REGION Network 26: Signal conditioning — Consolidate the auto or manual state request
   // ▀▀▀▀▀▀▀▀▀▀▀▀▀▀▀▀▀▀▀▀▀▀▀▀▀▀▀▀▀▀▀▀▀▀▀▀▀▀▀▀▀▀▀▀
   // Determine the valve state required by the automatic/manual mode selection:
   // 
   //    1.  If manual mode is active set wrkCtrlAutManOpCl to match the current manual 
   //      mode requested state (ctrl_Man_OpenClose)
   // 
   //    2.  If automatic mode is active set wrkCtrlAutManOpCl to match the current automatic 
   //      mode requested state (ctrl_Aut_OpenClose)
   // ▄▄▄▄▄▄▄▄▄▄▄▄▄▄▄▄▄▄▄▄▄▄▄▄▄▄▄▄▄▄▄▄▄▄▄▄▄▄▄▄▄▄▄▄
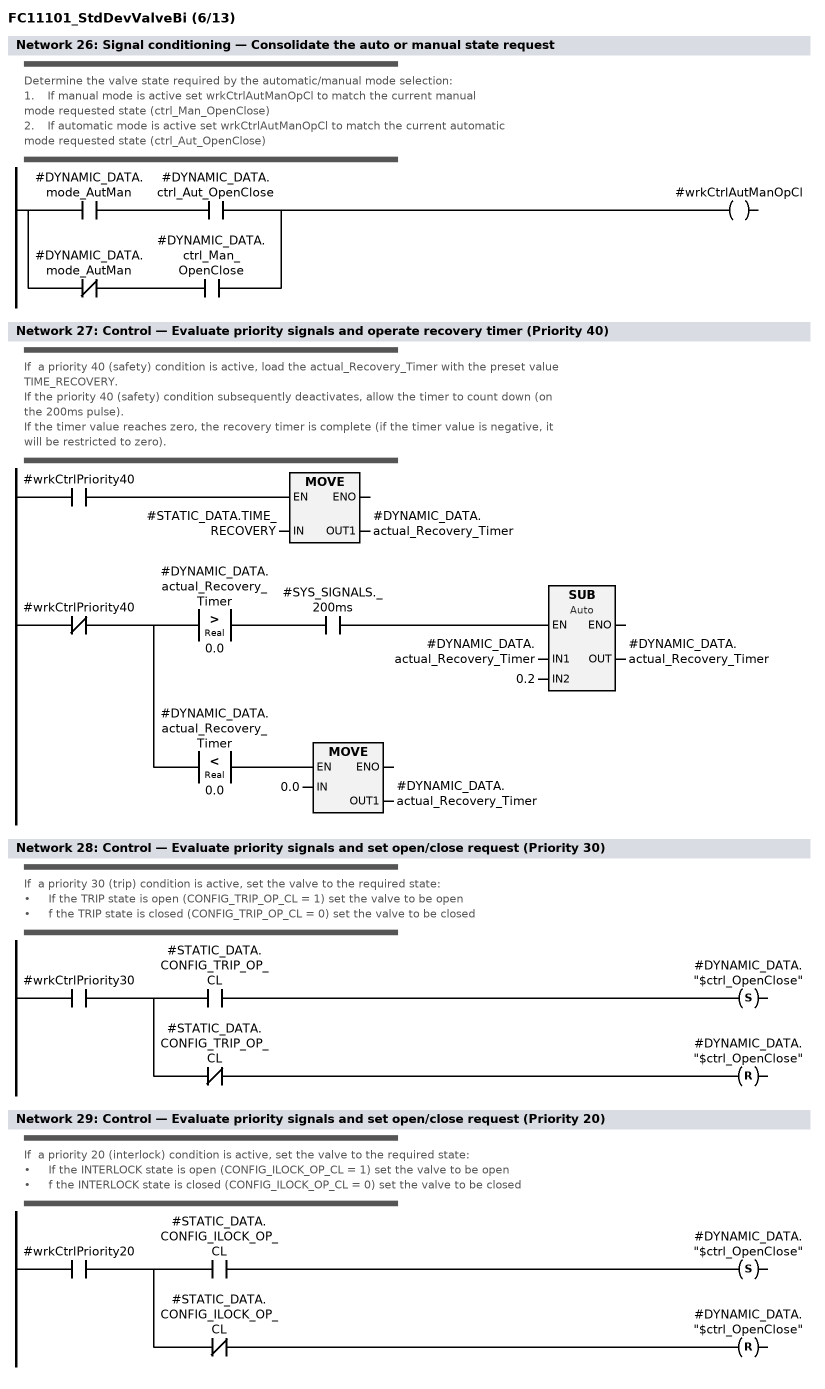
   RUNG wire#powerrail
      Contact( #DYNAMIC_DATA.mode_AutMan )
      Contact( #DYNAMIC_DATA.ctrl_Aut_OpenClose )
      wire#w1
      Coil( #wrkCtrlAutManOpCl )
   END_RUNG
   RUNG wire#powerrail
      I_Contact( #DYNAMIC_DATA.mode_AutMan )
      Contact( #DYNAMIC_DATA.ctrl_Man_OpenClose )
   END_RUNG wire#w1
   // the same network as SCL:
   #wrkCtrlAutManOpCl := (#DYNAMIC_DATA.mode_AutMan AND #DYNAMIC_DATA.ctrl_Aut_OpenClose) OR (NOT #DYNAMIC_DATA.mode_AutMan AND #DYNAMIC_DATA.ctrl_Man_OpenClose);
END_REGION

REGION Network 27: Control — Evaluate priority signals and operate recovery timer (Priority 40)
   // ▀▀▀▀▀▀▀▀▀▀▀▀▀▀▀▀▀▀▀▀▀▀▀▀▀▀▀▀▀▀▀▀▀▀▀▀▀▀▀▀▀▀▀▀
   // If  a priority 40 (safety) condition is active, load the actual_Recovery_Timer with the preset value 
   // TIME_RECOVERY.
   // 
   // If the priority 40 (safety) condition subsequently deactivates, allow the timer to count down (on 
   // the 200ms pulse).
   // 
   // If the timer value reaches zero, the recovery timer is complete (if the timer value is negative, it
   // will be restricted to zero).
   // ▄▄▄▄▄▄▄▄▄▄▄▄▄▄▄▄▄▄▄▄▄▄▄▄▄▄▄▄▄▄▄▄▄▄▄▄▄▄▄▄▄▄▄▄
   RUNG wire#powerrail
      Contact( #wrkCtrlPriority40 )
      Move(in := #STATIC_DATA.TIME_RECOVERY, out1 => #DYNAMIC_DATA.actual_Recovery_Timer)
   END_RUNG
   RUNG wire#powerrail
      I_Contact( #wrkCtrlPriority40 )
      wire#w1
      { S7_Templates := "SrcType := Real" } GT_Contact(in1 := #DYNAMIC_DATA.actual_Recovery_Timer, in2 := 0.0)
      Contact( #SYS_SIGNALS._200ms )
      Sub(in1 := #DYNAMIC_DATA.actual_Recovery_Timer, in2 := 0.2, out => #DYNAMIC_DATA.actual_Recovery_Timer)
   END_RUNG
   RUNG wire#w1
      { S7_Templates := "SrcType := Real" } LT_Contact(in1 := #DYNAMIC_DATA.actual_Recovery_Timer, in2 := 0.0)
      Move(in := 0.0, out1 => #DYNAMIC_DATA.actual_Recovery_Timer)
   END_RUNG
   // the same network as SCL:
   IF #wrkCtrlPriority40 THEN #DYNAMIC_DATA.actual_Recovery_Timer := #STATIC_DATA.TIME_RECOVERY; END_IF;
   IF NOT #wrkCtrlPriority40 AND (#DYNAMIC_DATA.actual_Recovery_Timer > 0.0) AND #SYS_SIGNALS._200ms THEN
       #DYNAMIC_DATA.actual_Recovery_Timer := #DYNAMIC_DATA.actual_Recovery_Timer - 0.2;
   END_IF;
   IF NOT #wrkCtrlPriority40 AND (#DYNAMIC_DATA.actual_Recovery_Timer < 0.0) THEN
       #DYNAMIC_DATA.actual_Recovery_Timer := 0.0;
   END_IF;
END_REGION

REGION Network 28: Control — Evaluate priority signals and set open/close request (Priority 30)
   // ▀▀▀▀▀▀▀▀▀▀▀▀▀▀▀▀▀▀▀▀▀▀▀▀▀▀▀▀▀▀▀▀▀▀▀▀▀▀▀▀▀▀▀▀
   // If  a priority 30 (trip) condition is active, set the valve to the required state:
   // 
   //    •   If the TRIP state is open (CONFIG_TRIP_OP_CL = 1) set the valve to be open
   // 
   //    •   f the TRIP state is closed (CONFIG_TRIP_OP_CL = 0) set the valve to be closed
   // ▄▄▄▄▄▄▄▄▄▄▄▄▄▄▄▄▄▄▄▄▄▄▄▄▄▄▄▄▄▄▄▄▄▄▄▄▄▄▄▄▄▄▄▄
   RUNG wire#powerrail
      Contact( #wrkCtrlPriority30 )
      wire#w1
      Contact( #STATIC_DATA.CONFIG_TRIP_OP_CL )
      S_Coil( #DYNAMIC_DATA."$ctrl_OpenClose" )
   END_RUNG
   RUNG wire#w1
      I_Contact( #STATIC_DATA.CONFIG_TRIP_OP_CL )
      R_Coil( #DYNAMIC_DATA."$ctrl_OpenClose" )
   END_RUNG
   // the same network as SCL:
   IF #wrkCtrlPriority30 AND #STATIC_DATA.CONFIG_TRIP_OP_CL THEN
       #DYNAMIC_DATA."$ctrl_OpenClose" := TRUE;
   END_IF;
   IF #wrkCtrlPriority30 AND NOT #STATIC_DATA.CONFIG_TRIP_OP_CL THEN
       #DYNAMIC_DATA."$ctrl_OpenClose" := FALSE;
   END_IF;
END_REGION

REGION Network 29: Control — Evaluate priority signals and set open/close request (Priority 20)
   // ▀▀▀▀▀▀▀▀▀▀▀▀▀▀▀▀▀▀▀▀▀▀▀▀▀▀▀▀▀▀▀▀▀▀▀▀▀▀▀▀▀▀▀▀
   // If  a priority 20 (interlock) condition is active, set the valve to the required state:
   // 
   //    •   If the INTERLOCK state is open (CONFIG_ILOCK_OP_CL = 1) set the valve to be open
   // 
   //    •   f the INTERLOCK state is closed (CONFIG_ILOCK_OP_CL = 0) set the valve to be closed
   // ▄▄▄▄▄▄▄▄▄▄▄▄▄▄▄▄▄▄▄▄▄▄▄▄▄▄▄▄▄▄▄▄▄▄▄▄▄▄▄▄▄▄▄▄
   RUNG wire#powerrail
      Contact( #wrkCtrlPriority20 )
      wire#w1
      Contact( #STATIC_DATA.CONFIG_ILOCK_OP_CL )
      S_Coil( #DYNAMIC_DATA."$ctrl_OpenClose" )
   END_RUNG
   RUNG wire#w1
      I_Contact( #STATIC_DATA.CONFIG_ILOCK_OP_CL )
      R_Coil( #DYNAMIC_DATA."$ctrl_OpenClose" )
   END_RUNG
   // the same network as SCL:
   IF #wrkCtrlPriority20 AND #STATIC_DATA.CONFIG_ILOCK_OP_CL THEN
       #DYNAMIC_DATA."$ctrl_OpenClose" := TRUE;
   END_IF;
   IF #wrkCtrlPriority20 AND NOT #STATIC_DATA.CONFIG_ILOCK_OP_CL THEN
       #DYNAMIC_DATA."$ctrl_OpenClose" := FALSE;
   END_IF;
END_REGION

REGION Network 30: Control — Evaluate priority signals and set open/close request (Priority 10)
   // ▀▀▀▀▀▀▀▀▀▀▀▀▀▀▀▀▀▀▀▀▀▀▀▀▀▀▀▀▀▀▀▀▀▀▀▀▀▀▀▀▀▀▀▀
   // If  a priority 10 (permissive) condition is active, set the valve to the required state:
   // 
   // 
   // PERMITTED STATE IS OPEN — CONDITIONS:
   // 
   //    •   If the Permitted state is open and Aut/Man request is for open, 
   //      set the valve to be open [Branch 1]
   // 
   //    •   If the Permitted state is open and Aut/Man request is for closed, and the current
   //      valve output matches this state (closed), set the valve to be closed (maintain the
   //      current state) [Branch 6]
   // 
   //    •   If the Permitted state is open and Aut/Man request is for closed, and the current
   //      valve output matches the open state, set the valve to be open (override the
   //      auto/man request [Branch 2]
   // 
   // PERMITTED STATE IS CLOSED — CONDITIONS:
   // 
   //    •   If the Permitted state is closed and Aut/Man request is for closed,
   //      set the valve to be  closed [Branch 4]
   // 
   //    •   If the Permitted state is closed and Aut/Man request is for open, and the current
   //      valve output matches this state (open), set the valve to be open (maintain the
   //      current state) [Branch 3]
   // 
   //    •   If the Permitted state is closed and Aut/Man request is for open, and the current
   //      valve output matches the closed state, set the valve to be closed (override the
   //      auto/man request [Branch 5]
   // ▄▄▄▄▄▄▄▄▄▄▄▄▄▄▄▄▄▄▄▄▄▄▄▄▄▄▄▄▄▄▄▄▄▄▄▄▄▄▄▄▄▄▄▄
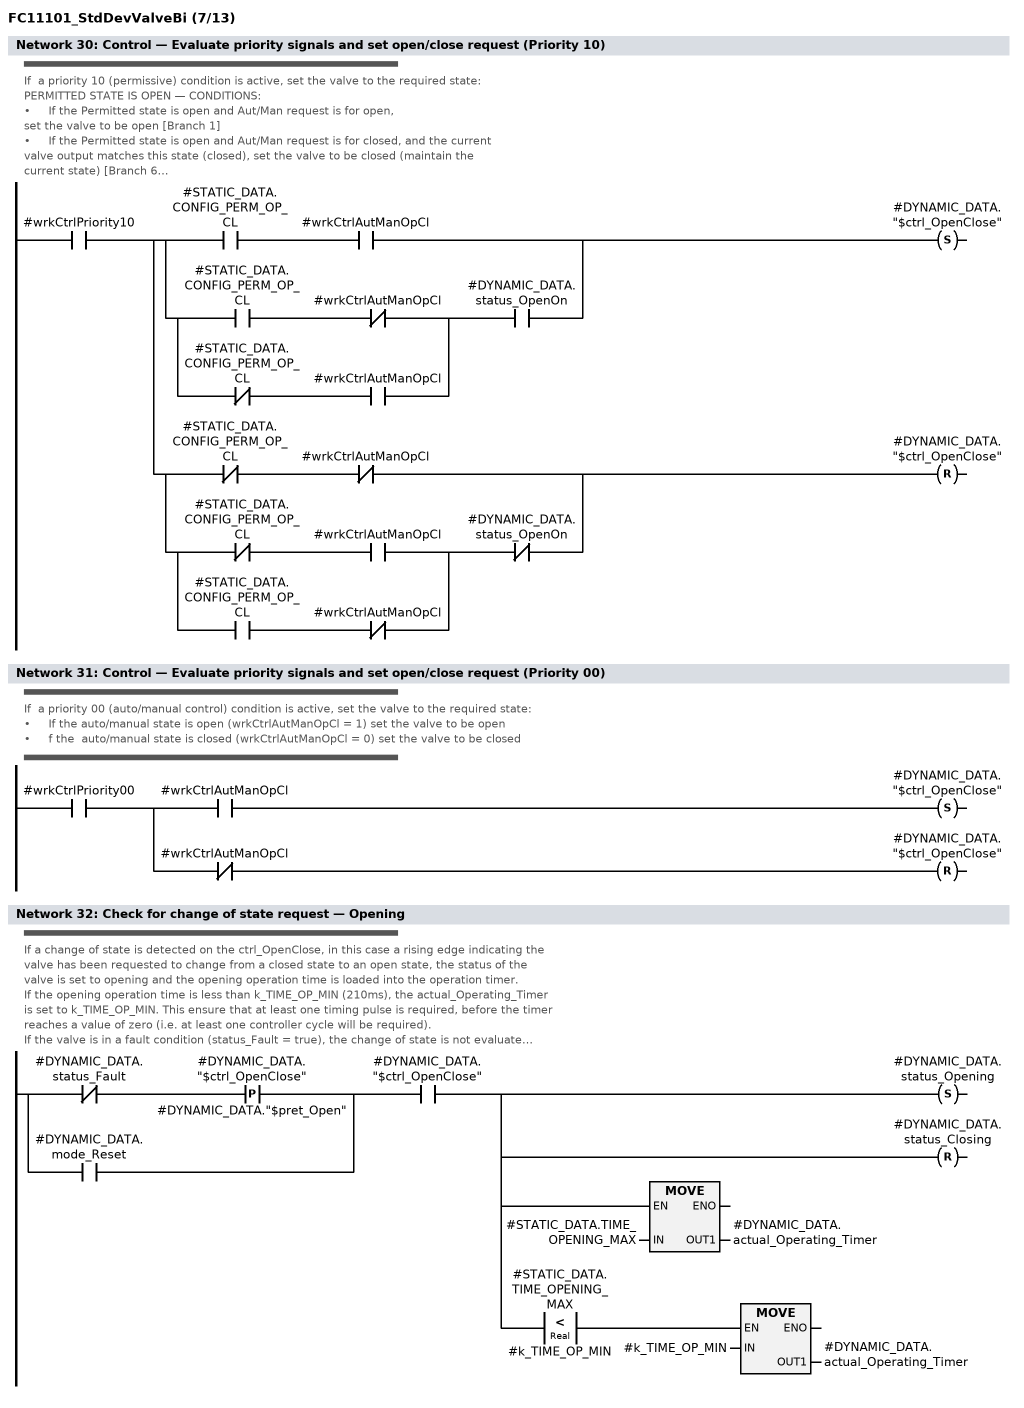
   RUNG wire#powerrail
      Contact( #wrkCtrlPriority10 )
      wire#w1
      Contact( #STATIC_DATA.CONFIG_PERM_OP_CL )
      Contact( #wrkCtrlAutManOpCl )
      wire#w2
      S_Coil( #DYNAMIC_DATA."$ctrl_OpenClose" )
   END_RUNG
   RUNG wire#w1
      Contact( #STATIC_DATA.CONFIG_PERM_OP_CL )
      I_Contact( #wrkCtrlAutManOpCl )
      wire#w3
      Contact( #DYNAMIC_DATA.status_OpenOn )
   END_RUNG wire#w2
   RUNG wire#w1
      I_Contact( #STATIC_DATA.CONFIG_PERM_OP_CL )
      Contact( #wrkCtrlAutManOpCl )
   END_RUNG wire#w3
   RUNG wire#w1
      I_Contact( #STATIC_DATA.CONFIG_PERM_OP_CL )
      I_Contact( #wrkCtrlAutManOpCl )
      wire#w4
      R_Coil( #DYNAMIC_DATA."$ctrl_OpenClose" )
   END_RUNG
   RUNG wire#w1
      I_Contact( #STATIC_DATA.CONFIG_PERM_OP_CL )
      Contact( #wrkCtrlAutManOpCl )
      wire#w5
      I_Contact( #DYNAMIC_DATA.status_OpenOn )
   END_RUNG wire#w4
   RUNG wire#w1
      Contact( #STATIC_DATA.CONFIG_PERM_OP_CL )
      I_Contact( #wrkCtrlAutManOpCl )
   END_RUNG wire#w5
   // the same network as SCL:
   IF #wrkCtrlPriority10 AND ((#STATIC_DATA.CONFIG_PERM_OP_CL AND #wrkCtrlAutManOpCl) OR (((#STATIC_DATA.CONFIG_PERM_OP_CL AND NOT #wrkCtrlAutManOpCl) OR (NOT #STATIC_DATA.CONFIG_PERM_OP_CL AND #wrkCtrlAutManOpCl)) AND #DYNAMIC_DATA.status_OpenOn)) THEN
       #DYNAMIC_DATA."$ctrl_OpenClose" := TRUE;
   END_IF;
   IF #wrkCtrlPriority10 AND ((NOT #STATIC_DATA.CONFIG_PERM_OP_CL AND NOT #wrkCtrlAutManOpCl) OR (((NOT #STATIC_DATA.CONFIG_PERM_OP_CL AND #wrkCtrlAutManOpCl) OR (#STATIC_DATA.CONFIG_PERM_OP_CL AND NOT #wrkCtrlAutManOpCl)) AND NOT #DYNAMIC_DATA.status_OpenOn)) THEN
       #DYNAMIC_DATA."$ctrl_OpenClose" := FALSE;
   END_IF;
END_REGION

REGION Network 31: Control — Evaluate priority signals and set open/close request (Priority 00)
   // ▀▀▀▀▀▀▀▀▀▀▀▀▀▀▀▀▀▀▀▀▀▀▀▀▀▀▀▀▀▀▀▀▀▀▀▀▀▀▀▀▀▀▀▀
   // If  a priority 00 (auto/manual control) condition is active, set the valve to the required state:
   // 
   //    •   If the auto/manual state is open (wrkCtrlAutManOpCl = 1) set the valve to be open
   // 
   //    •   f the  auto/manual state is closed (wrkCtrlAutManOpCl = 0) set the valve to be closed
   // ▄▄▄▄▄▄▄▄▄▄▄▄▄▄▄▄▄▄▄▄▄▄▄▄▄▄▄▄▄▄▄▄▄▄▄▄▄▄▄▄▄▄▄▄
   RUNG wire#powerrail
      Contact( #wrkCtrlPriority00 )
      wire#w1
      Contact( #wrkCtrlAutManOpCl )
      S_Coil( #DYNAMIC_DATA."$ctrl_OpenClose" )
   END_RUNG
   RUNG wire#w1
      I_Contact( #wrkCtrlAutManOpCl )
      R_Coil( #DYNAMIC_DATA."$ctrl_OpenClose" )
   END_RUNG
   // the same network as SCL:
   IF #wrkCtrlPriority00 AND #wrkCtrlAutManOpCl THEN #DYNAMIC_DATA."$ctrl_OpenClose" := TRUE; END_IF;
   IF #wrkCtrlPriority00 AND NOT #wrkCtrlAutManOpCl THEN #DYNAMIC_DATA."$ctrl_OpenClose" := FALSE; END_IF;
END_REGION

REGION Network 32: Check for change of state request — Opening
   // ▀▀▀▀▀▀▀▀▀▀▀▀▀▀▀▀▀▀▀▀▀▀▀▀▀▀▀▀▀▀▀▀▀▀▀▀▀▀▀▀▀▀▀▀
   // If a change of state is detected on the ctrl_OpenClose, in this case a rising edge indicating the
   // valve has been requested to change from a closed state to an open state, the status of the
   // valve is set to opening and the opening operation time is loaded into the operation timer.
   // 
   // If the opening operation time is less than k_TIME_OP_MIN (210ms), the actual_Operating_Timer 
   // is set to k_TIME_OP_MIN. This ensure that at least one timing pulse is required, before the timer 
   // reaches a value of zero (i.e. at least one controller cycle will be required).
   // 
   // If the valve is in a fault condition (status_Fault = true), the change of state is not evaluated
   // until the fault condition has cleared
   // 
   // Note: the timer is also triggered if the Reset signal is received and the valve is requested open.
   // ▄▄▄▄▄▄▄▄▄▄▄▄▄▄▄▄▄▄▄▄▄▄▄▄▄▄▄▄▄▄▄▄▄▄▄▄▄▄▄▄▄▄▄▄
   RUNG wire#powerrail
      I_Contact( #DYNAMIC_DATA.status_Fault )
      P_Contact(operand := #DYNAMIC_DATA."$ctrl_OpenClose", bit := #DYNAMIC_DATA."$pret_Open")
      wire#w1
      Contact( #DYNAMIC_DATA."$ctrl_OpenClose" )
      wire#w2
      S_Coil( #DYNAMIC_DATA.status_Opening )
   END_RUNG
   RUNG wire#powerrail
      Contact( #DYNAMIC_DATA.mode_Reset )
   END_RUNG wire#w1
   RUNG wire#w2
      R_Coil( #DYNAMIC_DATA.status_Closing )
   END_RUNG
   RUNG wire#w2
      Move(in := #STATIC_DATA.TIME_OPENING_MAX, out1 => #DYNAMIC_DATA.actual_Operating_Timer)
   END_RUNG
   RUNG wire#w2
      { S7_Templates := "SrcType := Real" } LT_Contact(in1 := #STATIC_DATA.TIME_OPENING_MAX, in2 := #k_TIME_OP_MIN)
      Move(in := #k_TIME_OP_MIN, out1 => #DYNAMIC_DATA.actual_Operating_Timer)
   END_RUNG
   // the same network as SCL:
   #_w1 := NOT #DYNAMIC_DATA.status_Fault AND #DYNAMIC_DATA."$ctrl_OpenClose" AND NOT #DYNAMIC_DATA."$pret_Open";   // rising edge of #DYNAMIC_DATA."$ctrl_OpenClose"
   #DYNAMIC_DATA."$pret_Open" := #DYNAMIC_DATA."$ctrl_OpenClose";
   #_w2 := (#_w1 OR #DYNAMIC_DATA.mode_Reset) AND #DYNAMIC_DATA."$ctrl_OpenClose";
   IF #_w2 THEN
       #DYNAMIC_DATA.status_Opening := TRUE;
       #DYNAMIC_DATA.status_Closing := FALSE;
       #DYNAMIC_DATA.actual_Operating_Timer := #STATIC_DATA.TIME_OPENING_MAX;
   END_IF;
   IF #_w2 AND (#STATIC_DATA.TIME_OPENING_MAX < #k_TIME_OP_MIN) THEN
       #DYNAMIC_DATA.actual_Operating_Timer := #k_TIME_OP_MIN;
   END_IF;
END_REGION

REGION Network 33: Check for change of state request — Closing
   // ▀▀▀▀▀▀▀▀▀▀▀▀▀▀▀▀▀▀▀▀▀▀▀▀▀▀▀▀▀▀▀▀▀▀▀▀▀▀▀▀▀▀▀▀
   // If a change of state is detected on the ctrl_OpenClose, in this case a falling edge indicating the
   // valve has been requested to change from an open state to a closed state, the status of the
   // valve is set to closing and the closing operation time is loaded into the operation timer.
   // 
   // If the closing operation time is less than k_TIME_OP_MIN (210ms), the actual_Operating_Timer 
   // is set to k_TIME_OP_MIN. This ensure that at least one timing pulse is required, before the timer 
   // reaches a value of zero (i.e. at least one controller cycle will be required).
   // 
   // If the valve is in a fault condition (status_Fault = true), the change of state is not evaluated
   // until the fault condition has cleared
   // 
   // Note: the timer is also triggered if the Reset signal is received and the valve is requested closed.
   // ▄▄▄▄▄▄▄▄▄▄▄▄▄▄▄▄▄▄▄▄▄▄▄▄▄▄▄▄▄▄▄▄▄▄▄▄▄▄▄▄▄▄▄▄
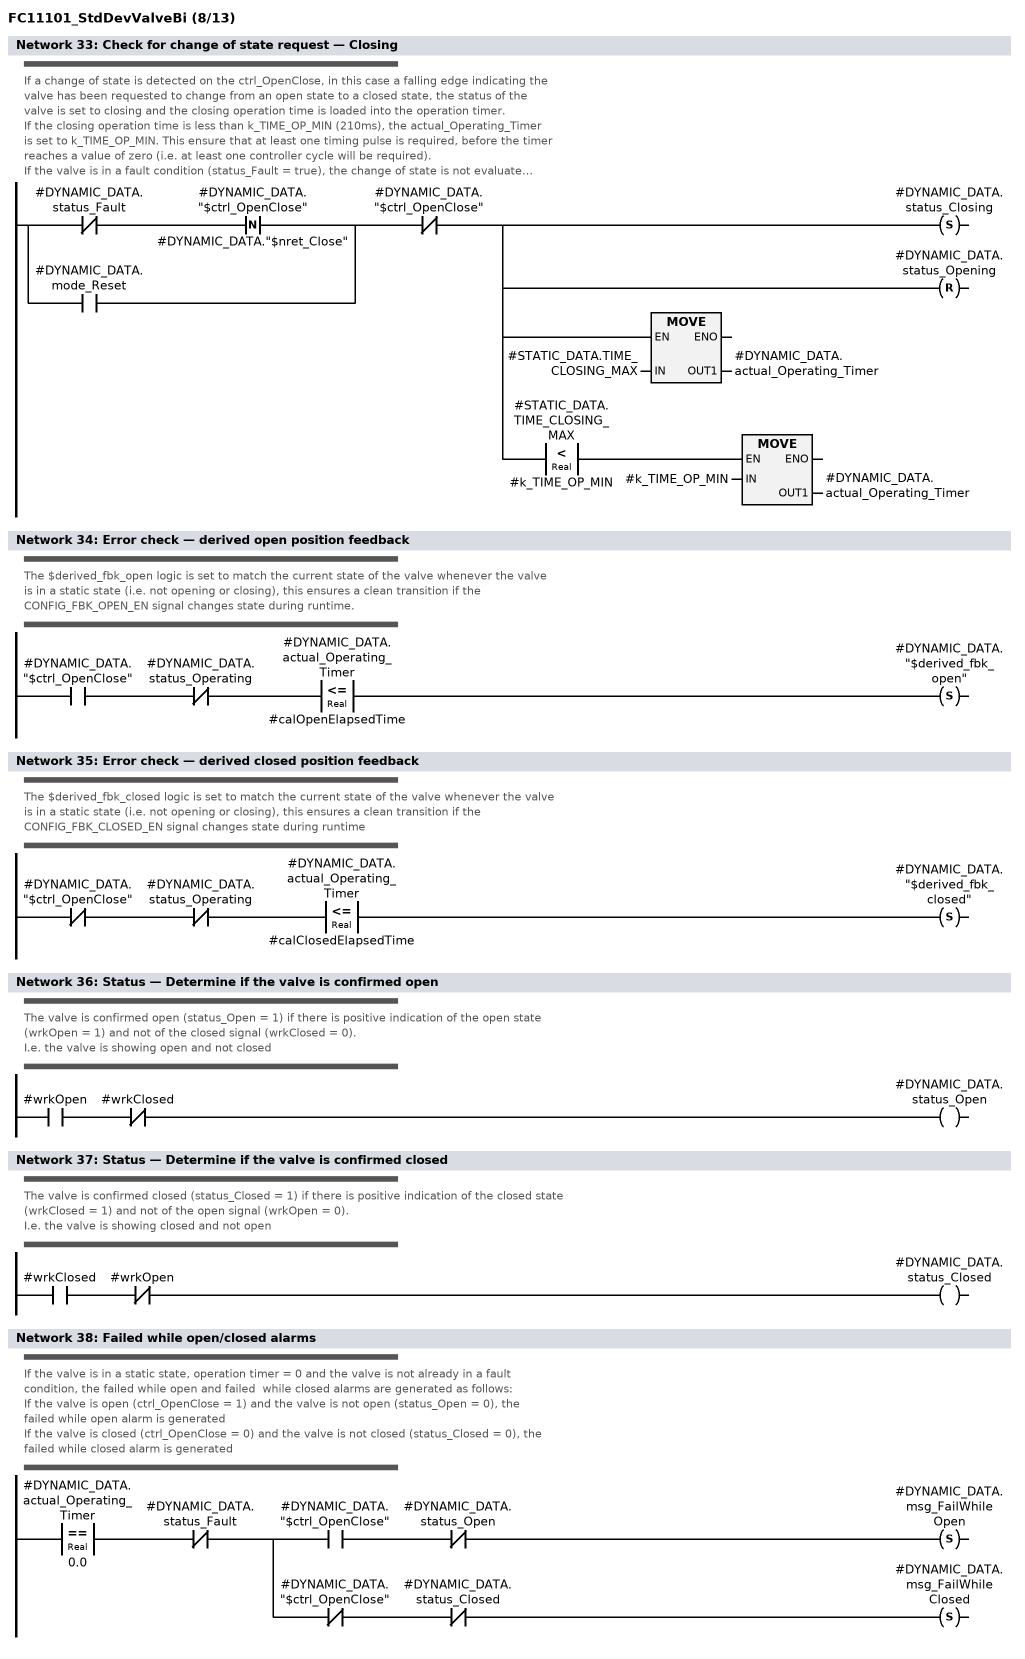
   RUNG wire#powerrail
      I_Contact( #DYNAMIC_DATA.status_Fault )
      N_Contact(operand := #DYNAMIC_DATA."$ctrl_OpenClose", bit := #DYNAMIC_DATA."$nret_Close")
      wire#w1
      I_Contact( #DYNAMIC_DATA."$ctrl_OpenClose" )
      wire#w2
      S_Coil( #DYNAMIC_DATA.status_Closing )
   END_RUNG
   RUNG wire#powerrail
      Contact( #DYNAMIC_DATA.mode_Reset )
   END_RUNG wire#w1
   RUNG wire#w2
      R_Coil( #DYNAMIC_DATA.status_Opening )
   END_RUNG
   RUNG wire#w2
      Move(in := #STATIC_DATA.TIME_CLOSING_MAX, out1 => #DYNAMIC_DATA.actual_Operating_Timer)
   END_RUNG
   RUNG wire#w2
      { S7_Templates := "SrcType := Real" } LT_Contact(in1 := #STATIC_DATA.TIME_CLOSING_MAX, in2 := #k_TIME_OP_MIN)
      Move(in := #k_TIME_OP_MIN, out1 => #DYNAMIC_DATA.actual_Operating_Timer)
   END_RUNG
   // the same network as SCL:
   #_w1 := NOT #DYNAMIC_DATA.status_Fault AND NOT #DYNAMIC_DATA."$ctrl_OpenClose" AND #DYNAMIC_DATA."$nret_Close";   // falling edge of #DYNAMIC_DATA."$ctrl_OpenClose"
   #DYNAMIC_DATA."$nret_Close" := #DYNAMIC_DATA."$ctrl_OpenClose";
   #_w2 := (#_w1 OR #DYNAMIC_DATA.mode_Reset) AND NOT #DYNAMIC_DATA."$ctrl_OpenClose";
   IF #_w2 THEN
       #DYNAMIC_DATA.status_Closing := TRUE;
       #DYNAMIC_DATA.status_Opening := FALSE;
       #DYNAMIC_DATA.actual_Operating_Timer := #STATIC_DATA.TIME_CLOSING_MAX;
   END_IF;
   IF #_w2 AND (#STATIC_DATA.TIME_CLOSING_MAX < #k_TIME_OP_MIN) THEN
       #DYNAMIC_DATA.actual_Operating_Timer := #k_TIME_OP_MIN;
   END_IF;
END_REGION

REGION Network 34: Error check — derived open position feedback
   // ▀▀▀▀▀▀▀▀▀▀▀▀▀▀▀▀▀▀▀▀▀▀▀▀▀▀▀▀▀▀▀▀▀▀▀▀▀▀▀▀▀▀▀▀
   // The $derived_fbk_open logic is set to match the current state of the valve whenever the valve
   // is in a static state (i.e. not opening or closing), this ensures a clean transition if the 
   // CONFIG_FBK_OPEN_EN signal changes state during runtime.
   // ▄▄▄▄▄▄▄▄▄▄▄▄▄▄▄▄▄▄▄▄▄▄▄▄▄▄▄▄▄▄▄▄▄▄▄▄▄▄▄▄▄▄▄▄
   RUNG wire#powerrail
      Contact( #DYNAMIC_DATA."$ctrl_OpenClose" )
      I_Contact( #DYNAMIC_DATA.status_Operating )
      { S7_Templates := "SrcType := Real" } LE_Contact(in1 := #DYNAMIC_DATA.actual_Operating_Timer, in2 := #calOpenElapsedTime)
      S_Coil( #DYNAMIC_DATA."$derived_fbk_open" )
   END_RUNG
   // the same network as SCL:
   IF #DYNAMIC_DATA."$ctrl_OpenClose" AND NOT #DYNAMIC_DATA.status_Operating AND (#DYNAMIC_DATA.actual_Operating_Timer <= #calOpenElapsedTime) THEN
       #DYNAMIC_DATA."$derived_fbk_open" := TRUE;
   END_IF;
END_REGION

REGION Network 35: Error check — derived closed position feedback
   // ▀▀▀▀▀▀▀▀▀▀▀▀▀▀▀▀▀▀▀▀▀▀▀▀▀▀▀▀▀▀▀▀▀▀▀▀▀▀▀▀▀▀▀▀
   // The $derived_fbk_closed logic is set to match the current state of the valve whenever the valve
   // is in a static state (i.e. not opening or closing), this ensures a clean transition if the 
   // CONFIG_FBK_CLOSED_EN signal changes state during runtime
   // ▄▄▄▄▄▄▄▄▄▄▄▄▄▄▄▄▄▄▄▄▄▄▄▄▄▄▄▄▄▄▄▄▄▄▄▄▄▄▄▄▄▄▄▄
   RUNG wire#powerrail
      I_Contact( #DYNAMIC_DATA."$ctrl_OpenClose" )
      I_Contact( #DYNAMIC_DATA.status_Operating )
      { S7_Templates := "SrcType := Real" } LE_Contact(in1 := #DYNAMIC_DATA.actual_Operating_Timer, in2 := #calClosedElapsedTime)
      S_Coil( #DYNAMIC_DATA."$derived_fbk_closed" )
   END_RUNG
   // the same network as SCL:
   IF NOT #DYNAMIC_DATA."$ctrl_OpenClose" AND NOT #DYNAMIC_DATA.status_Operating AND (#DYNAMIC_DATA.actual_Operating_Timer <= #calClosedElapsedTime) THEN
       #DYNAMIC_DATA."$derived_fbk_closed" := TRUE;
   END_IF;
END_REGION

REGION Network 36: Status — Determine if the valve is confirmed open
   // ▀▀▀▀▀▀▀▀▀▀▀▀▀▀▀▀▀▀▀▀▀▀▀▀▀▀▀▀▀▀▀▀▀▀▀▀▀▀▀▀▀▀▀▀
   // The valve is confirmed open (status_Open = 1) if there is positive indication of the open state 
   // (wrkOpen = 1) and not of the closed signal (wrkClosed = 0). 
   // 
   // I.e. the valve is showing open and not closed
   // ▄▄▄▄▄▄▄▄▄▄▄▄▄▄▄▄▄▄▄▄▄▄▄▄▄▄▄▄▄▄▄▄▄▄▄▄▄▄▄▄▄▄▄▄
   RUNG wire#powerrail
      Contact( #wrkOpen )
      I_Contact( #wrkClosed )
      Coil( #DYNAMIC_DATA.status_Open )
   END_RUNG
   // the same network as SCL:
   #DYNAMIC_DATA.status_Open := #wrkOpen AND NOT #wrkClosed;
END_REGION

REGION Network 37: Status — Determine if the valve is confirmed closed
   // ▀▀▀▀▀▀▀▀▀▀▀▀▀▀▀▀▀▀▀▀▀▀▀▀▀▀▀▀▀▀▀▀▀▀▀▀▀▀▀▀▀▀▀▀
   // The valve is confirmed closed (status_Closed = 1) if there is positive indication of the closed state 
   // (wrkClosed = 1) and not of the open signal (wrkOpen = 0). 
   // 
   // I.e. the valve is showing closed and not open
   // ▄▄▄▄▄▄▄▄▄▄▄▄▄▄▄▄▄▄▄▄▄▄▄▄▄▄▄▄▄▄▄▄▄▄▄▄▄▄▄▄▄▄▄▄
   RUNG wire#powerrail
      Contact( #wrkClosed )
      I_Contact( #wrkOpen )
      Coil( #DYNAMIC_DATA.status_Closed )
   END_RUNG
   // the same network as SCL:
   #DYNAMIC_DATA.status_Closed := #wrkClosed AND NOT #wrkOpen;
END_REGION

REGION Network 38: Failed while open/closed alarms
   // ▀▀▀▀▀▀▀▀▀▀▀▀▀▀▀▀▀▀▀▀▀▀▀▀▀▀▀▀▀▀▀▀▀▀▀▀▀▀▀▀▀▀▀▀
   // If the valve is in a static state, operation timer = 0 and the valve is not already in a fault
   // condition, the failed while open and failed  while closed alarms are generated as follows:
   // 
   // If the valve is open (ctrl_OpenClose = 1) and the valve is not open (status_Open = 0), the 
   // failed while open alarm is generated
   // 
   // If the valve is closed (ctrl_OpenClose = 0) and the valve is not closed (status_Closed = 0), the 
   // failed while closed alarm is generated
   // ▄▄▄▄▄▄▄▄▄▄▄▄▄▄▄▄▄▄▄▄▄▄▄▄▄▄▄▄▄▄▄▄▄▄▄▄▄▄▄▄▄▄▄▄
   RUNG wire#powerrail
      { S7_Templates := "SrcType := Real" } EQ_Contact(in1 := #DYNAMIC_DATA.actual_Operating_Timer, in2 := 0.0)
      I_Contact( #DYNAMIC_DATA.status_Fault )
      wire#w1
      Contact( #DYNAMIC_DATA."$ctrl_OpenClose" )
      I_Contact( #DYNAMIC_DATA.status_Open )
      S_Coil( #DYNAMIC_DATA.msg_FailWhileOpen )
   END_RUNG
   RUNG wire#w1
      I_Contact( #DYNAMIC_DATA."$ctrl_OpenClose" )
      I_Contact( #DYNAMIC_DATA.status_Closed )
      S_Coil( #DYNAMIC_DATA.msg_FailWhileClosed )
   END_RUNG
   // the same network as SCL:
   #_w1 := (#DYNAMIC_DATA.actual_Operating_Timer = 0.0) AND NOT #DYNAMIC_DATA.status_Fault;
   IF #_w1 AND #DYNAMIC_DATA."$ctrl_OpenClose" AND NOT #DYNAMIC_DATA.status_Open THEN
       #DYNAMIC_DATA.msg_FailWhileOpen := TRUE;
   END_IF;
   IF #_w1 AND NOT #DYNAMIC_DATA."$ctrl_OpenClose" AND NOT #DYNAMIC_DATA.status_Closed THEN
       #DYNAMIC_DATA.msg_FailWhileClosed := TRUE;
   END_IF;
END_REGION

REGION Network 39: Operation timer and Failed to open/close alarms
   // ▀▀▀▀▀▀▀▀▀▀▀▀▀▀▀▀▀▀▀▀▀▀▀▀▀▀▀▀▀▀▀▀▀▀▀▀▀▀▀▀▀▀▀▀
   // If the valve is opening or closing, decrement the current operation timer value on each 200ms
   // pulse.
   // 
   // If the timer reaches zero, and the valve is opening, generate the failed to open alarm.
   // 
   // If the timer reaches zero, and the valve is closing, generate the failed to close alarm
   // ▄▄▄▄▄▄▄▄▄▄▄▄▄▄▄▄▄▄▄▄▄▄▄▄▄▄▄▄▄▄▄▄▄▄▄▄▄▄▄▄▄▄▄▄
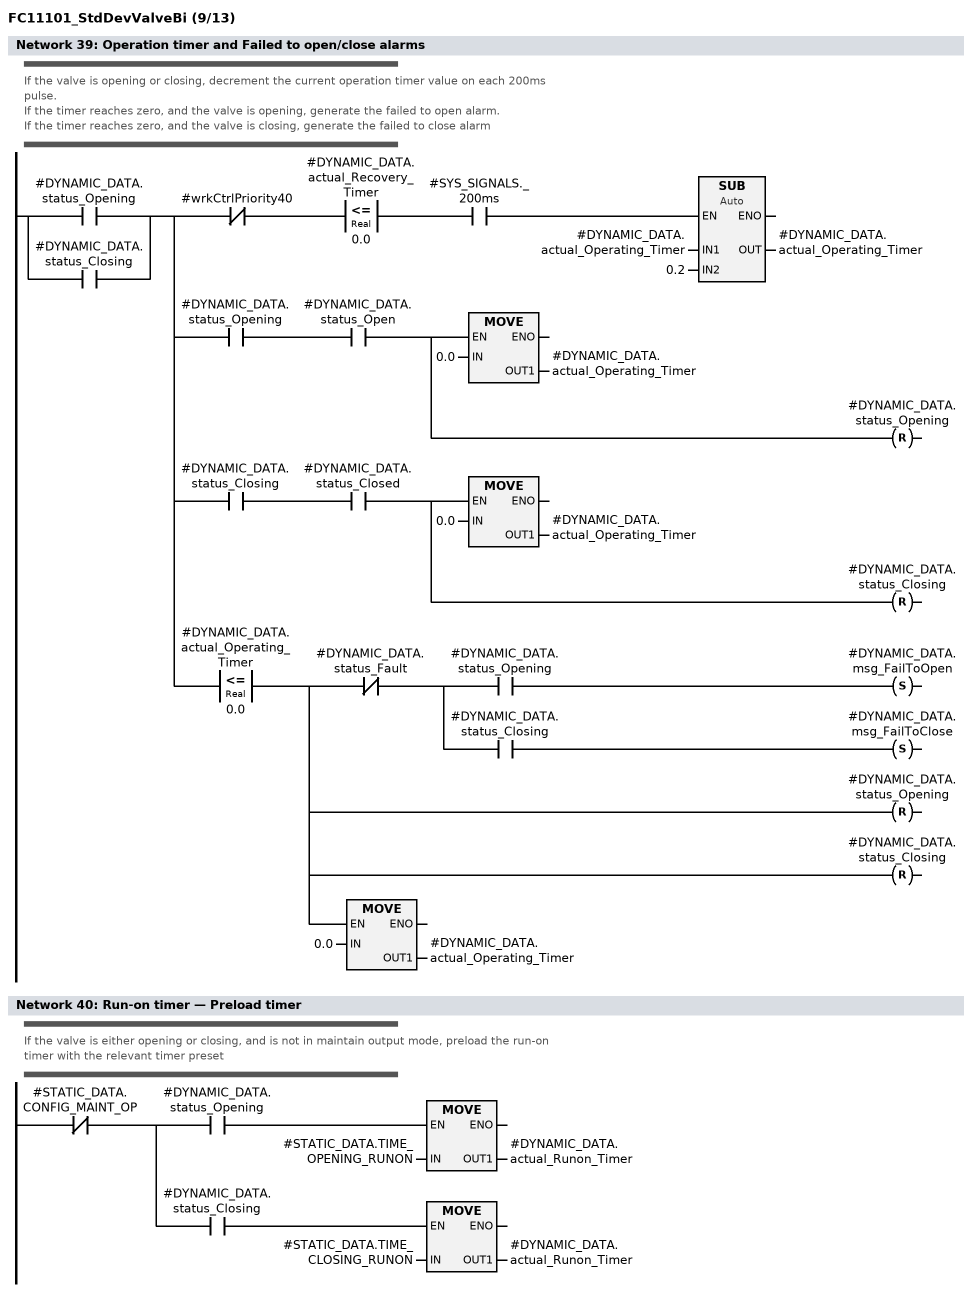
   RUNG wire#powerrail
      Contact( #DYNAMIC_DATA.status_Opening )
      wire#w1
      I_Contact( #wrkCtrlPriority40 )
      { S7_Templates := "SrcType := Real" } LE_Contact(in1 := #DYNAMIC_DATA.actual_Recovery_Timer, in2 := 0.0)
      Contact( #SYS_SIGNALS._200ms )
      Sub(in1 := #DYNAMIC_DATA.actual_Operating_Timer, in2 := 0.2, out => #DYNAMIC_DATA.actual_Operating_Timer)
   END_RUNG
   RUNG wire#powerrail
      Contact( #DYNAMIC_DATA.status_Closing )
   END_RUNG wire#w1
   RUNG wire#w1
      Contact( #DYNAMIC_DATA.status_Opening )
      Contact( #DYNAMIC_DATA.status_Open )
      wire#w2
      Move(in := 0.0, out1 => #DYNAMIC_DATA.actual_Operating_Timer)
   END_RUNG
   RUNG wire#w2
      R_Coil( #DYNAMIC_DATA.status_Opening )
   END_RUNG
   RUNG wire#w1
      Contact( #DYNAMIC_DATA.status_Closing )
      Contact( #DYNAMIC_DATA.status_Closed )
      wire#w3
      Move(in := 0.0, out1 => #DYNAMIC_DATA.actual_Operating_Timer)
   END_RUNG
   RUNG wire#w3
      R_Coil( #DYNAMIC_DATA.status_Closing )
   END_RUNG
   RUNG wire#w1
      { S7_Templates := "SrcType := Real" } LE_Contact(in1 := #DYNAMIC_DATA.actual_Operating_Timer, in2 := 0.0)
      wire#w4
      I_Contact( #DYNAMIC_DATA.status_Fault )
      wire#w5
      Contact( #DYNAMIC_DATA.status_Opening )
      S_Coil( #DYNAMIC_DATA.msg_FailToOpen )
   END_RUNG
   RUNG wire#w5
      Contact( #DYNAMIC_DATA.status_Closing )
      S_Coil( #DYNAMIC_DATA.msg_FailToClose )
   END_RUNG
   RUNG wire#w4
      R_Coil( #DYNAMIC_DATA.status_Opening )
   END_RUNG
   RUNG wire#w4
      R_Coil( #DYNAMIC_DATA.status_Closing )
   END_RUNG
   RUNG wire#w4
      Move(in := 0.0, out1 => #DYNAMIC_DATA.actual_Operating_Timer)
   END_RUNG
   // the same network as SCL:
   #_w1 := #DYNAMIC_DATA.status_Opening OR #DYNAMIC_DATA.status_Closing;
   IF #_w1 AND NOT #wrkCtrlPriority40 AND (#DYNAMIC_DATA.actual_Recovery_Timer <= 0.0) AND #SYS_SIGNALS._200ms THEN
       #DYNAMIC_DATA.actual_Operating_Timer := #DYNAMIC_DATA.actual_Operating_Timer - 0.2;
   END_IF;
   IF #_w1 AND #DYNAMIC_DATA.status_Opening AND #DYNAMIC_DATA.status_Open THEN
       #DYNAMIC_DATA.actual_Operating_Timer := 0.0;
       #DYNAMIC_DATA.status_Opening := FALSE;
   END_IF;
   IF #_w1 AND #DYNAMIC_DATA.status_Closing AND #DYNAMIC_DATA.status_Closed THEN
       #DYNAMIC_DATA.actual_Operating_Timer := 0.0;
       #DYNAMIC_DATA.status_Closing := FALSE;
   END_IF;
   #_w2 := #_w1 AND (#DYNAMIC_DATA.actual_Operating_Timer <= 0.0);
   #_w3 := #_w2 AND NOT #DYNAMIC_DATA.status_Fault;
   IF #_w3 AND #DYNAMIC_DATA.status_Opening THEN #DYNAMIC_DATA.msg_FailToOpen := TRUE; END_IF;
   IF #_w3 AND #DYNAMIC_DATA.status_Closing THEN #DYNAMIC_DATA.msg_FailToClose := TRUE; END_IF;
   IF #_w2 THEN
       #DYNAMIC_DATA.status_Opening := FALSE;
       #DYNAMIC_DATA.status_Closing := FALSE;
       #DYNAMIC_DATA.actual_Operating_Timer := 0.0;
   END_IF;
END_REGION

REGION Network 40: Run-on timer — Preload timer
   // ▀▀▀▀▀▀▀▀▀▀▀▀▀▀▀▀▀▀▀▀▀▀▀▀▀▀▀▀▀▀▀▀▀▀▀▀▀▀▀▀▀▀▀▀
   // If the valve is either opening or closing, and is not in maintain output mode, preload the run-on
   // timer with the relevant timer preset
   // ▄▄▄▄▄▄▄▄▄▄▄▄▄▄▄▄▄▄▄▄▄▄▄▄▄▄▄▄▄▄▄▄▄▄▄▄▄▄▄▄▄▄▄▄
   RUNG wire#powerrail
      I_Contact( #STATIC_DATA.CONFIG_MAINT_OP )
      wire#w1
      Contact( #DYNAMIC_DATA.status_Opening )
      Move(in := #STATIC_DATA.TIME_OPENING_RUNON, out1 => #DYNAMIC_DATA.actual_Runon_Timer)
   END_RUNG
   RUNG wire#w1
      Contact( #DYNAMIC_DATA.status_Closing )
      Move(in := #STATIC_DATA.TIME_CLOSING_RUNON, out1 => #DYNAMIC_DATA.actual_Runon_Timer)
   END_RUNG
   // the same network as SCL:
   #_w1 := NOT #STATIC_DATA.CONFIG_MAINT_OP;
   IF #_w1 AND #DYNAMIC_DATA.status_Opening THEN
       #DYNAMIC_DATA.actual_Runon_Timer := #STATIC_DATA.TIME_OPENING_RUNON;
   END_IF;
   IF #_w1 AND #DYNAMIC_DATA.status_Closing THEN
       #DYNAMIC_DATA.actual_Runon_Timer := #STATIC_DATA.TIME_CLOSING_RUNON;
   END_IF;
END_REGION

REGION Network 41: Run-on timer — Count down
   // ▀▀▀▀▀▀▀▀▀▀▀▀▀▀▀▀▀▀▀▀▀▀▀▀▀▀▀▀▀▀▀▀▀▀▀▀▀▀▀▀▀▀▀▀
   // If the valve is either closed or open, is not in fault and is not configured to maintain outputs, the 
   // run-on timer will count down from its preset value.
   // 
   // If an emergency stop is activated whilst the run-on timer is active, it will pause at the last 
   // elapsed value.
   // 
   // If a fault condition is active or if the valve is configured to maintain outputs, the run-on timer is
   // set to zero.
   // ▄▄▄▄▄▄▄▄▄▄▄▄▄▄▄▄▄▄▄▄▄▄▄▄▄▄▄▄▄▄▄▄▄▄▄▄▄▄▄▄▄▄▄▄
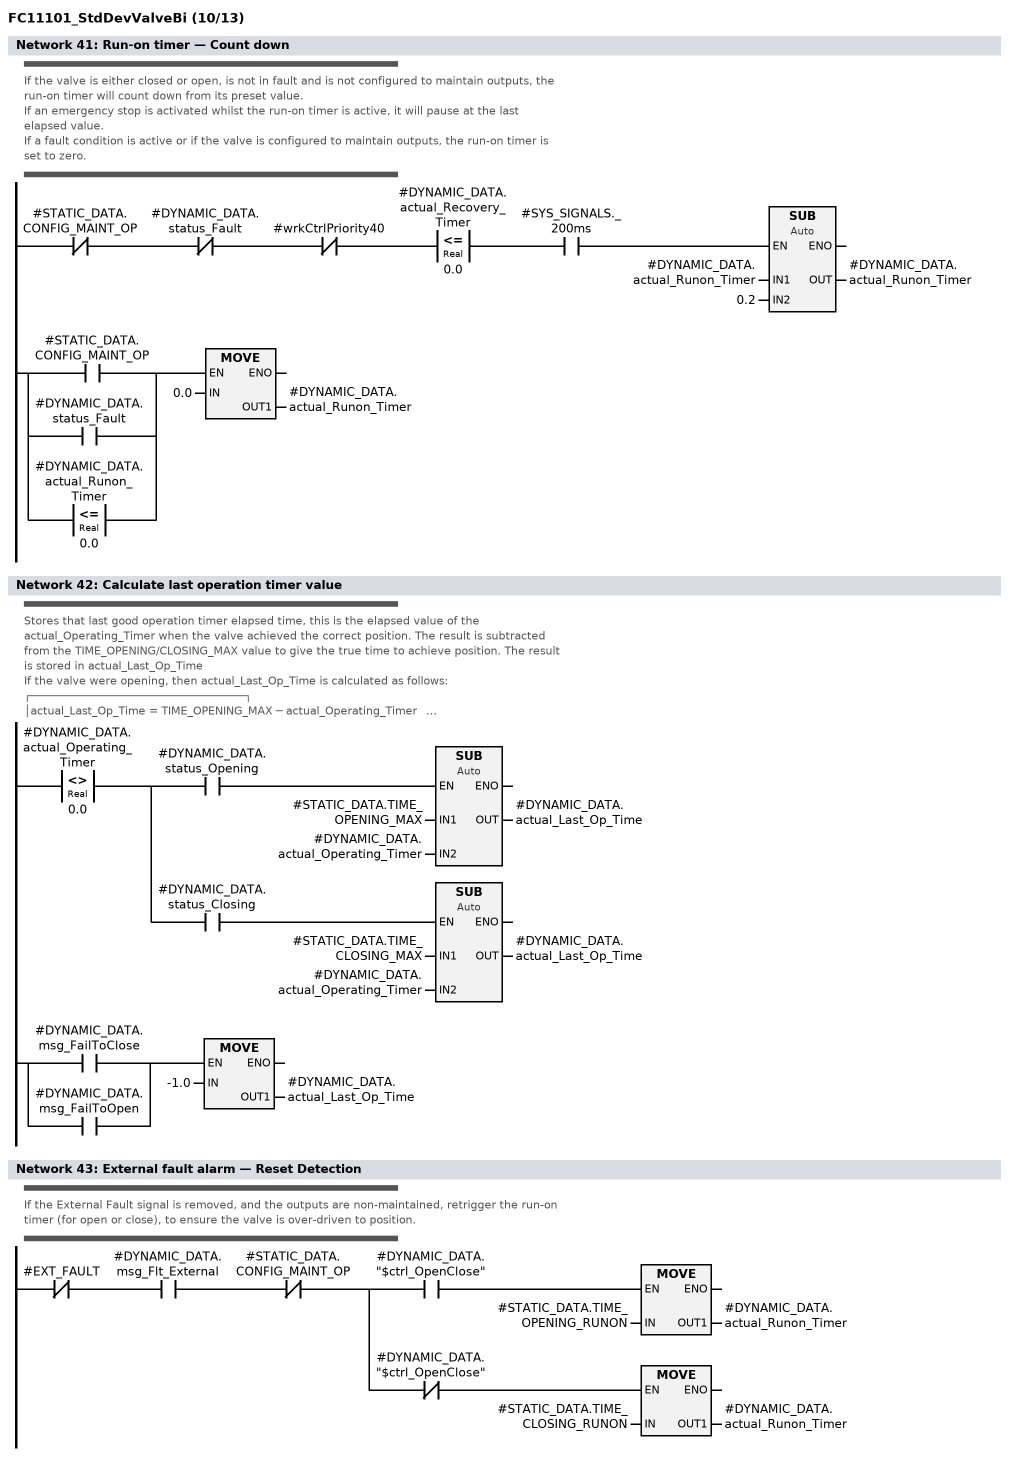
   RUNG wire#powerrail
      I_Contact( #STATIC_DATA.CONFIG_MAINT_OP )
      I_Contact( #DYNAMIC_DATA.status_Fault )
      I_Contact( #wrkCtrlPriority40 )
      { S7_Templates := "SrcType := Real" } LE_Contact(in1 := #DYNAMIC_DATA.actual_Recovery_Timer, in2 := 0.0)
      Contact( #SYS_SIGNALS._200ms )
      Sub(in1 := #DYNAMIC_DATA.actual_Runon_Timer, in2 := 0.2, out => #DYNAMIC_DATA.actual_Runon_Timer)
   END_RUNG
   RUNG wire#powerrail
      Contact( #STATIC_DATA.CONFIG_MAINT_OP )
      wire#w1
      Move(in := 0.0, out1 => #DYNAMIC_DATA.actual_Runon_Timer)
   END_RUNG
   RUNG wire#powerrail
      Contact( #DYNAMIC_DATA.status_Fault )
   END_RUNG wire#w1
   RUNG wire#powerrail
      { S7_Templates := "SrcType := Real" } LE_Contact(in1 := #DYNAMIC_DATA.actual_Runon_Timer, in2 := 0.0)
   END_RUNG wire#w1
   // the same network as SCL:
   IF NOT #STATIC_DATA.CONFIG_MAINT_OP AND NOT #DYNAMIC_DATA.status_Fault AND NOT #wrkCtrlPriority40 AND (#DYNAMIC_DATA.actual_Recovery_Timer <= 0.0) AND #SYS_SIGNALS._200ms THEN
       #DYNAMIC_DATA.actual_Runon_Timer := #DYNAMIC_DATA.actual_Runon_Timer - 0.2;
   END_IF;
   IF #STATIC_DATA.CONFIG_MAINT_OP OR #DYNAMIC_DATA.status_Fault OR (#DYNAMIC_DATA.actual_Runon_Timer <= 0.0) THEN
       #DYNAMIC_DATA.actual_Runon_Timer := 0.0;
   END_IF;
END_REGION

REGION Network 42: Calculate last operation timer value
   // ▀▀▀▀▀▀▀▀▀▀▀▀▀▀▀▀▀▀▀▀▀▀▀▀▀▀▀▀▀▀▀▀▀▀▀▀▀▀▀▀▀▀▀▀
   // Stores that last good operation timer elapsed time, this is the elapsed value of the 
   // actual_Operating_Timer when the valve achieved the correct position. The result is subtracted
   // from the TIME_OPENING/CLOSING_MAX value to give the true time to achieve position. The result
   // is stored in actual_Last_Op_Time
   // 
   // If the valve were opening, then actual_Last_Op_Time is calculated as follows:
   // 
   // ┌─────────────────────────────────┐
   // │actual_Last_Op_Time = TIME_OPENING_MAX ─ actual_Operating_Timer   │
   // └─────────────────────────────────┘
   // 
   // If the valve were closing, then actual_Last_Op_Time is calculated as follows:
   // 
   // ┌─────────────────────────────────┐
   // │actual_Last_Op_Time = TIME_CLOSING_MAX ─ actual_Operating_Timer   │
   // └─────────────────────────────────┘
   // 
   // If the valve either fails to open or fails to close,  then actual_Last_Op_Time is set to -1.0 to 
   // indicate a fault state.
   // ▄▄▄▄▄▄▄▄▄▄▄▄▄▄▄▄▄▄▄▄▄▄▄▄▄▄▄▄▄▄▄▄▄▄▄▄▄▄▄▄▄▄▄▄
   RUNG wire#powerrail
      { S7_Templates := "SrcType := Real" } NE_Contact(in1 := #DYNAMIC_DATA.actual_Operating_Timer, in2 := 0.0)
      wire#w1
      Contact( #DYNAMIC_DATA.status_Opening )
      Sub(in1 := #STATIC_DATA.TIME_OPENING_MAX, in2 := #DYNAMIC_DATA.actual_Operating_Timer, out => #DYNAMIC_DATA.actual_Last_Op_Time)
   END_RUNG
   RUNG wire#w1
      Contact( #DYNAMIC_DATA.status_Closing )
      Sub(in1 := #STATIC_DATA.TIME_CLOSING_MAX, in2 := #DYNAMIC_DATA.actual_Operating_Timer, out => #DYNAMIC_DATA.actual_Last_Op_Time)
   END_RUNG
   RUNG wire#powerrail
      Contact( #DYNAMIC_DATA.msg_FailToClose )
      wire#w2
      Move(in := -1.0, out1 => #DYNAMIC_DATA.actual_Last_Op_Time)
   END_RUNG
   RUNG wire#powerrail
      Contact( #DYNAMIC_DATA.msg_FailToOpen )
   END_RUNG wire#w2
   // the same network as SCL:
   #_w1 := #DYNAMIC_DATA.actual_Operating_Timer <> 0.0;
   IF #_w1 AND #DYNAMIC_DATA.status_Opening THEN
       #DYNAMIC_DATA.actual_Last_Op_Time := #STATIC_DATA.TIME_OPENING_MAX - #DYNAMIC_DATA.actual_Operating_Timer;
   END_IF;
   IF #_w1 AND #DYNAMIC_DATA.status_Closing THEN
       #DYNAMIC_DATA.actual_Last_Op_Time := #STATIC_DATA.TIME_CLOSING_MAX - #DYNAMIC_DATA.actual_Operating_Timer;
   END_IF;
   IF #DYNAMIC_DATA.msg_FailToClose OR #DYNAMIC_DATA.msg_FailToOpen THEN
       #DYNAMIC_DATA.actual_Last_Op_Time := -1.0;
   END_IF;
END_REGION

REGION Network 43: External fault alarm — Reset Detection
   // ▀▀▀▀▀▀▀▀▀▀▀▀▀▀▀▀▀▀▀▀▀▀▀▀▀▀▀▀▀▀▀▀▀▀▀▀▀▀▀▀▀▀▀▀
   // If the External Fault signal is removed, and the outputs are non-maintained, retrigger the run-on 
   // timer (for open or close), to ensure the valve is over-driven to position.
   // ▄▄▄▄▄▄▄▄▄▄▄▄▄▄▄▄▄▄▄▄▄▄▄▄▄▄▄▄▄▄▄▄▄▄▄▄▄▄▄▄▄▄▄▄
   RUNG wire#powerrail
      I_Contact( #EXT_FAULT )
      Contact( #DYNAMIC_DATA.msg_Flt_External )
      I_Contact( #STATIC_DATA.CONFIG_MAINT_OP )
      wire#w1
      Contact( #DYNAMIC_DATA."$ctrl_OpenClose" )
      Move(in := #STATIC_DATA.TIME_OPENING_RUNON, out1 => #DYNAMIC_DATA.actual_Runon_Timer)
   END_RUNG
   RUNG wire#w1
      I_Contact( #DYNAMIC_DATA."$ctrl_OpenClose" )
      Move(in := #STATIC_DATA.TIME_CLOSING_RUNON, out1 => #DYNAMIC_DATA.actual_Runon_Timer)
   END_RUNG
   // the same network as SCL:
   #_w1 := NOT #EXT_FAULT AND #DYNAMIC_DATA.msg_Flt_External AND NOT #STATIC_DATA.CONFIG_MAINT_OP;
   IF #_w1 AND #DYNAMIC_DATA."$ctrl_OpenClose" THEN
       #DYNAMIC_DATA.actual_Runon_Timer := #STATIC_DATA.TIME_OPENING_RUNON;
   END_IF;
   IF #_w1 AND NOT #DYNAMIC_DATA."$ctrl_OpenClose" THEN
       #DYNAMIC_DATA.actual_Runon_Timer := #STATIC_DATA.TIME_CLOSING_RUNON;
   END_IF;
END_REGION

REGION Network 44: External fault alarm
   // ▀▀▀▀▀▀▀▀▀▀▀▀▀▀▀▀▀▀▀▀▀▀▀▀▀▀▀▀▀▀▀▀▀▀▀▀▀▀▀▀▀▀▀▀
   // If the external fault signal (EXT_FAULT) is active, generate the external fault alarm
   // ▄▄▄▄▄▄▄▄▄▄▄▄▄▄▄▄▄▄▄▄▄▄▄▄▄▄▄▄▄▄▄▄▄▄▄▄▄▄▄▄▄▄▄▄
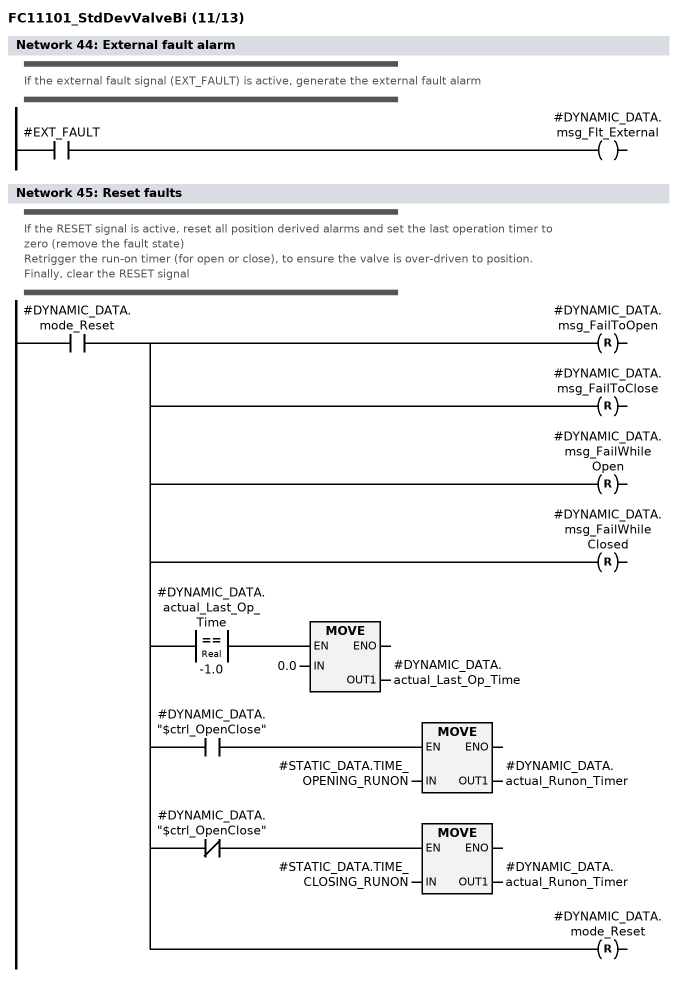
   RUNG wire#powerrail
      Contact( #EXT_FAULT )
      Coil( #DYNAMIC_DATA.msg_Flt_External )
   END_RUNG
   // the same network as SCL:
   #DYNAMIC_DATA.msg_Flt_External := #EXT_FAULT;
END_REGION

REGION Network 45: Reset faults
   // ▀▀▀▀▀▀▀▀▀▀▀▀▀▀▀▀▀▀▀▀▀▀▀▀▀▀▀▀▀▀▀▀▀▀▀▀▀▀▀▀▀▀▀▀
   // If the RESET signal is active, reset all position derived alarms and set the last operation timer to
   // zero (remove the fault state)
   // 
   // Retrigger the run-on timer (for open or close), to ensure the valve is over-driven to position.
   // 
   // Finally, clear the RESET signal
   // ▄▄▄▄▄▄▄▄▄▄▄▄▄▄▄▄▄▄▄▄▄▄▄▄▄▄▄▄▄▄▄▄▄▄▄▄▄▄▄▄▄▄▄▄
   RUNG wire#powerrail
      Contact( #DYNAMIC_DATA.mode_Reset )
      wire#w1
      R_Coil( #DYNAMIC_DATA.msg_FailToOpen )
   END_RUNG
   RUNG wire#w1
      R_Coil( #DYNAMIC_DATA.msg_FailToClose )
   END_RUNG
   RUNG wire#w1
      R_Coil( #DYNAMIC_DATA.msg_FailWhileOpen )
   END_RUNG
   RUNG wire#w1
      R_Coil( #DYNAMIC_DATA.msg_FailWhileClosed )
   END_RUNG
   RUNG wire#w1
      { S7_Templates := "SrcType := Real" } EQ_Contact(in1 := #DYNAMIC_DATA.actual_Last_Op_Time, in2 := -1.0)
      Move(in := 0.0, out1 => #DYNAMIC_DATA.actual_Last_Op_Time)
   END_RUNG
   RUNG wire#w1
      Contact( #DYNAMIC_DATA."$ctrl_OpenClose" )
      Move(in := #STATIC_DATA.TIME_OPENING_RUNON, out1 => #DYNAMIC_DATA.actual_Runon_Timer)
   END_RUNG
   RUNG wire#w1
      I_Contact( #DYNAMIC_DATA."$ctrl_OpenClose" )
      Move(in := #STATIC_DATA.TIME_CLOSING_RUNON, out1 => #DYNAMIC_DATA.actual_Runon_Timer)
   END_RUNG
   RUNG wire#w1
      R_Coil( #DYNAMIC_DATA.mode_Reset )
   END_RUNG
   // the same network as SCL:
   IF #DYNAMIC_DATA.mode_Reset THEN
       #DYNAMIC_DATA.msg_FailToOpen := FALSE;
       #DYNAMIC_DATA.msg_FailToClose := FALSE;
       #DYNAMIC_DATA.msg_FailWhileOpen := FALSE;
       #DYNAMIC_DATA.msg_FailWhileClosed := FALSE;
   END_IF;
   IF #DYNAMIC_DATA.mode_Reset AND (#DYNAMIC_DATA.actual_Last_Op_Time = (-1.0)) THEN
       #DYNAMIC_DATA.actual_Last_Op_Time := 0.0;
   END_IF;
   IF #DYNAMIC_DATA.mode_Reset AND #DYNAMIC_DATA."$ctrl_OpenClose" THEN
       #DYNAMIC_DATA.actual_Runon_Timer := #STATIC_DATA.TIME_OPENING_RUNON;
   END_IF;
   IF #DYNAMIC_DATA.mode_Reset AND NOT #DYNAMIC_DATA."$ctrl_OpenClose" THEN
       #DYNAMIC_DATA.actual_Runon_Timer := #STATIC_DATA.TIME_CLOSING_RUNON;
   END_IF;
   IF #DYNAMIC_DATA.mode_Reset THEN #DYNAMIC_DATA.mode_Reset := FALSE; END_IF;
END_REGION

REGION Network 46: Status signals
   // ▀▀▀▀▀▀▀▀▀▀▀▀▀▀▀▀▀▀▀▀▀▀▀▀▀▀▀▀▀▀▀▀▀▀▀▀▀▀▀▀▀▀▀▀
   // The status signals for faults, alarms and warnings are either duplicates of the message signals 
   // (signals beginning with msg_) or logical combinations of them.
   // 
   // The following is a full list of the status signals:
   // 
   //  UT31101_Dy_DevValveBi (full contents)
   //  ――――――――――――――――――――――――――――――――――――――――――
   //  SIGNAL NAME          FUNCTION                     TYPE
   //  ――――――――――――――――――――――――――――――――――――――――――
   //  status_Operating        STATUS — Valve is changing state           Bool
   //                      (1 = changing state, 0 = fixed state)
   //  status_Fault            STATUS — Valve is in fault              Bool
   //                      (1 = fault present, 0 = healthy)
   //  status_Energised        STATUS — Valve output is on              Bool
   //                      (1 = energised, 0 = deenergised)
   //  status_Aut           STATUS — Automatic mode active           Bool
   //                      (1 = auto mode on, 0 = auto mode off)
   //  status_Man          STATUS — Manual mode active             Bool
   //                      (1 = man mode on, 0 = man mode off)
   //  status_EStop          STATUS — E_STOP safety signal is active         Bool
   //                      (1 = active, 0 = healthy)
   //  status_Trip        STATUS — TRIP signal is active             Bool
   //                      (1 = active, 0 = healthy)
   //  status_Ilock         STATUS — INTERLOCK signal is active            Bool
   //                      (1 = active, 0 = healthy)
   //  status_Perm        STATUS — PERMISSIVE signal is active           Bool
   //                      (1 = active, 0 = healthy)
   //  status_BypassOn        STATUS — Valve is in bypass mode          Bool
   //                      (1 = Simulation mode, 0 = normal)
   //  status_SimOn           STATUS — Valve is in simulation mode               Bool
   //                      (1 = Simulation mode, 0 = normal)
   //  status_RemoteOn       STATUS — Valve is in remote mode                  Bool
   //                      (1 = Remote mode, 0 = normal)
   //  status_LocalOn         STATUS — Valve is in local mode                    Bool
   //                      (1 = Local mode, 0 = normal)
   //  status_RLOff         STATUS — Valve is in ALL mode                   Bool
   //                      (1 = ALL mode, 0 = normal)
   //  ――――――――――――――――――――――――――――――――――――――――――
   // ▄▄▄▄▄▄▄▄▄▄▄▄▄▄▄▄▄▄▄▄▄▄▄▄▄▄▄▄▄▄▄▄▄▄▄▄▄▄▄▄▄▄▄▄
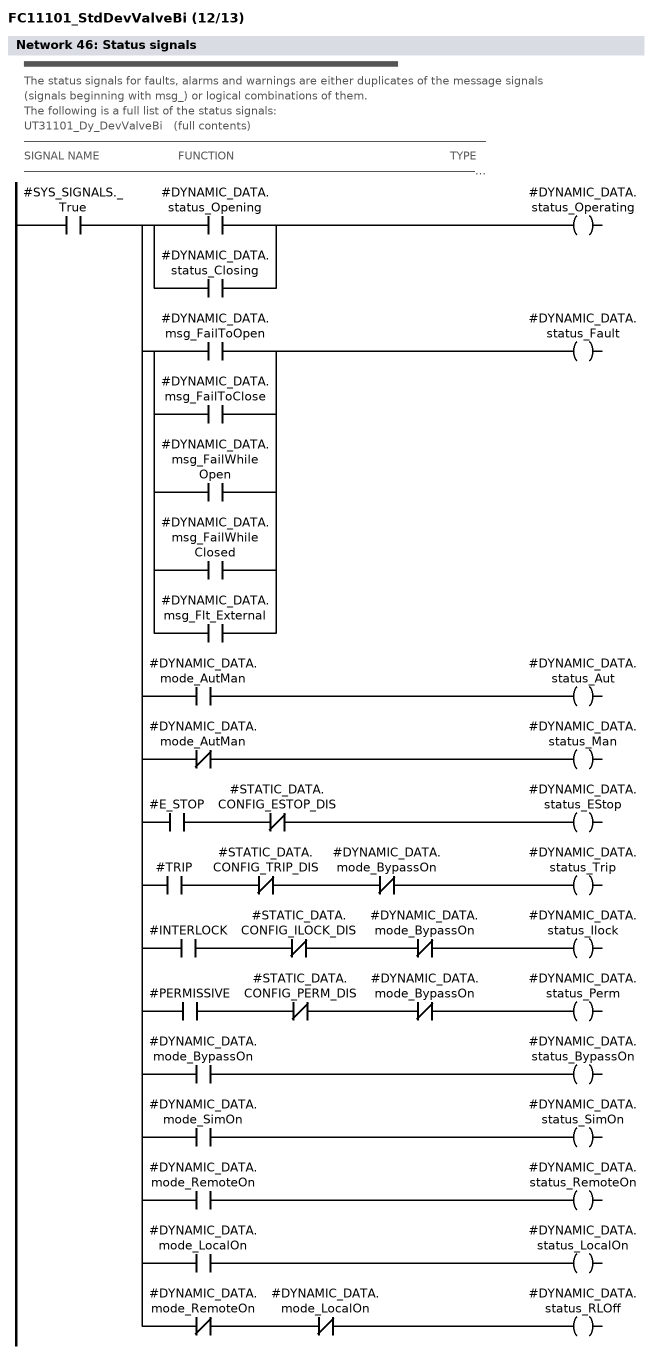
   RUNG wire#powerrail
      Contact( #SYS_SIGNALS._True )
      wire#w1
      Contact( #DYNAMIC_DATA.status_Opening )
      wire#w2
      Coil( #DYNAMIC_DATA.status_Operating )
   END_RUNG
   RUNG wire#w1
      Contact( #DYNAMIC_DATA.status_Closing )
   END_RUNG wire#w2
   RUNG wire#w1
      Contact( #DYNAMIC_DATA.msg_FailToOpen )
      wire#w3
      Coil( #DYNAMIC_DATA.status_Fault )
   END_RUNG
   RUNG wire#w1
      Contact( #DYNAMIC_DATA.msg_FailToClose )
   END_RUNG wire#w3
   RUNG wire#w1
      Contact( #DYNAMIC_DATA.msg_FailWhileOpen )
   END_RUNG wire#w3
   RUNG wire#w1
      Contact( #DYNAMIC_DATA.msg_FailWhileClosed )
   END_RUNG wire#w3
   RUNG wire#w1
      Contact( #DYNAMIC_DATA.msg_Flt_External )
   END_RUNG wire#w3
   RUNG wire#w1
      Contact( #DYNAMIC_DATA.mode_AutMan )
      Coil( #DYNAMIC_DATA.status_Aut )
   END_RUNG
   RUNG wire#w1
      I_Contact( #DYNAMIC_DATA.mode_AutMan )
      Coil( #DYNAMIC_DATA.status_Man )
   END_RUNG
   RUNG wire#w1
      Contact( #E_STOP )
      I_Contact( #STATIC_DATA.CONFIG_ESTOP_DIS )
      Coil( #DYNAMIC_DATA.status_EStop )
   END_RUNG
   RUNG wire#w1
      Contact( #TRIP )
      I_Contact( #STATIC_DATA.CONFIG_TRIP_DIS )
      I_Contact( #DYNAMIC_DATA.mode_BypassOn )
      Coil( #DYNAMIC_DATA.status_Trip )
   END_RUNG
   RUNG wire#w1
      Contact( #INTERLOCK )
      I_Contact( #STATIC_DATA.CONFIG_ILOCK_DIS )
      I_Contact( #DYNAMIC_DATA.mode_BypassOn )
      Coil( #DYNAMIC_DATA.status_Ilock )
   END_RUNG
   RUNG wire#w1
      Contact( #PERMISSIVE )
      I_Contact( #STATIC_DATA.CONFIG_PERM_DIS )
      I_Contact( #DYNAMIC_DATA.mode_BypassOn )
      Coil( #DYNAMIC_DATA.status_Perm )
   END_RUNG
   RUNG wire#w1
      Contact( #DYNAMIC_DATA.mode_BypassOn )
      Coil( #DYNAMIC_DATA.status_BypassOn )
   END_RUNG
   RUNG wire#w1
      Contact( #DYNAMIC_DATA.mode_SimOn )
      Coil( #DYNAMIC_DATA.status_SimOn )
   END_RUNG
   RUNG wire#w1
      Contact( #DYNAMIC_DATA.mode_RemoteOn )
      Coil( #DYNAMIC_DATA.status_RemoteOn )
   END_RUNG
   RUNG wire#w1
      Contact( #DYNAMIC_DATA.mode_LocalOn )
      Coil( #DYNAMIC_DATA.status_LocalOn )
   END_RUNG
   RUNG wire#w1
      I_Contact( #DYNAMIC_DATA.mode_RemoteOn )
      I_Contact( #DYNAMIC_DATA.mode_LocalOn )
      Coil( #DYNAMIC_DATA.status_RLOff )
   END_RUNG
   // the same network as SCL:
   #DYNAMIC_DATA.status_Operating := #SYS_SIGNALS._True AND (#DYNAMIC_DATA.status_Opening OR #DYNAMIC_DATA.status_Closing);
   #DYNAMIC_DATA.status_Fault := #SYS_SIGNALS._True AND (#DYNAMIC_DATA.msg_FailToOpen OR #DYNAMIC_DATA.msg_FailToClose OR #DYNAMIC_DATA.msg_FailWhileOpen OR #DYNAMIC_DATA.msg_FailWhileClosed OR #DYNAMIC_DATA.msg_Flt_External);
   #DYNAMIC_DATA.status_Aut := #SYS_SIGNALS._True AND #DYNAMIC_DATA.mode_AutMan;
   #DYNAMIC_DATA.status_Man := #SYS_SIGNALS._True AND NOT #DYNAMIC_DATA.mode_AutMan;
   #DYNAMIC_DATA.status_EStop := #SYS_SIGNALS._True AND #E_STOP AND NOT #STATIC_DATA.CONFIG_ESTOP_DIS;
   #DYNAMIC_DATA.status_Trip := #SYS_SIGNALS._True AND #TRIP AND NOT #STATIC_DATA.CONFIG_TRIP_DIS AND NOT #DYNAMIC_DATA.mode_BypassOn;
   #DYNAMIC_DATA.status_Ilock := #SYS_SIGNALS._True AND #INTERLOCK AND NOT #STATIC_DATA.CONFIG_ILOCK_DIS AND NOT #DYNAMIC_DATA.mode_BypassOn;
   #DYNAMIC_DATA.status_Perm := #SYS_SIGNALS._True AND #PERMISSIVE AND NOT #STATIC_DATA.CONFIG_PERM_DIS AND NOT #DYNAMIC_DATA.mode_BypassOn;
   #DYNAMIC_DATA.status_BypassOn := #SYS_SIGNALS._True AND #DYNAMIC_DATA.mode_BypassOn;
   #DYNAMIC_DATA.status_SimOn := #SYS_SIGNALS._True AND #DYNAMIC_DATA.mode_SimOn;
   #DYNAMIC_DATA.status_RemoteOn := #SYS_SIGNALS._True AND #DYNAMIC_DATA.mode_RemoteOn;
   #DYNAMIC_DATA.status_LocalOn := #SYS_SIGNALS._True AND #DYNAMIC_DATA.mode_LocalOn;
   #DYNAMIC_DATA.status_RLOff := #SYS_SIGNALS._True AND NOT #DYNAMIC_DATA.mode_RemoteOn AND NOT #DYNAMIC_DATA.mode_LocalOn;
END_REGION

REGION Network 47: OPEN_CMD output driver
   // ▀▀▀▀▀▀▀▀▀▀▀▀▀▀▀▀▀▀▀▀▀▀▀▀▀▀▀▀▀▀▀▀▀▀▀▀▀▀▀▀▀▀▀▀
   // The OPEN_CMD output drive will activate if all the following are true:
   // 
   //    1.  ESTOP is healthy or disabled (#wrkCtrlPriority40 = 1)
   // 
   //    2.  There is no fault condition (status_Fault = 0)
   // 
   //    3.  The valve is requested open ($ctrl_OpenClose = 1)
   // 
   //    4. The valve is opening (status_Opening =1)
   //         OR
   //      The valve is open (status_Open = 1) and either the run-on timer is active
   //      or the valve is configured to maintain outputs (CONFIG_MAINT_OP = 1)
   // 
   // The status_OpenOn signal is set to match the state of the OPEN_CMD
   // ▄▄▄▄▄▄▄▄▄▄▄▄▄▄▄▄▄▄▄▄▄▄▄▄▄▄▄▄▄▄▄▄▄▄▄▄▄▄▄▄▄▄▄▄
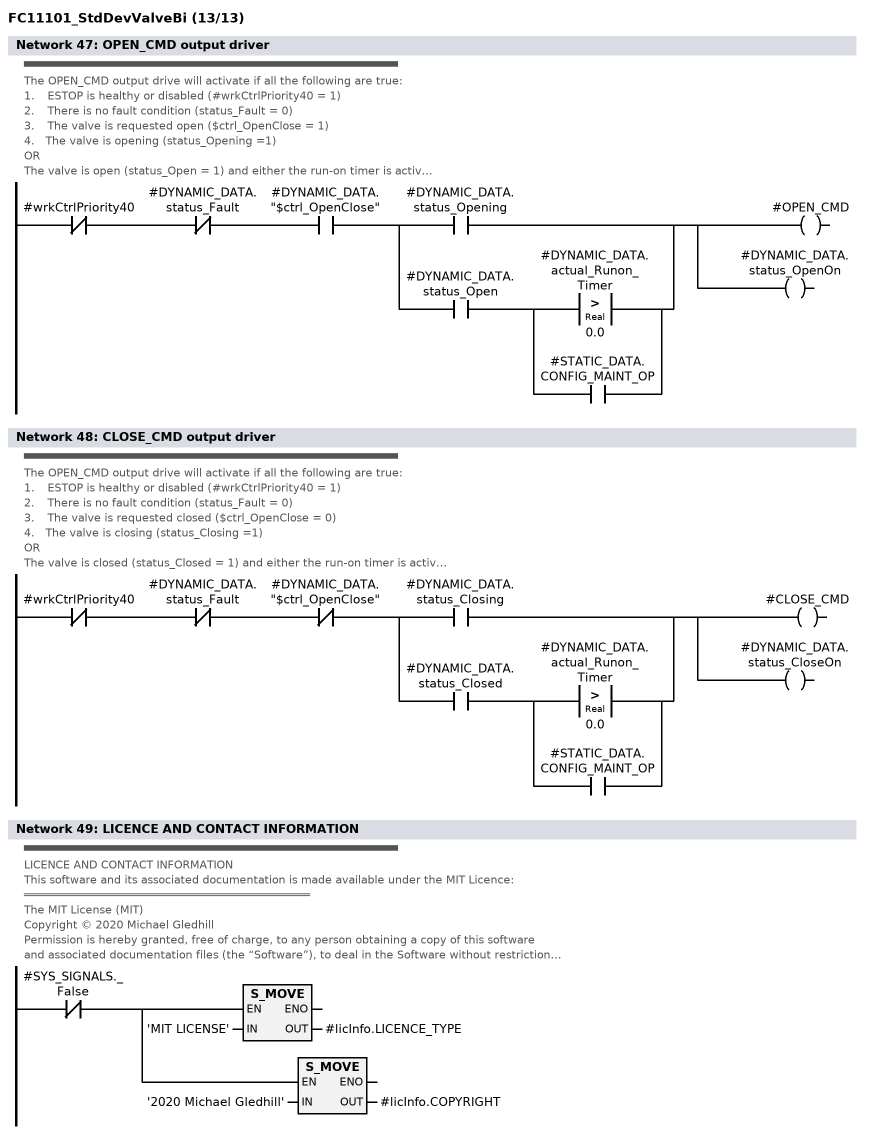
   RUNG wire#powerrail
      I_Contact( #wrkCtrlPriority40 )
      I_Contact( #DYNAMIC_DATA.status_Fault )
      Contact( #DYNAMIC_DATA."$ctrl_OpenClose" )
      wire#w1
      Contact( #DYNAMIC_DATA.status_Opening )
      wire#w2
      Coil( #OPEN_CMD )
   END_RUNG
   RUNG wire#w1
      Contact( #DYNAMIC_DATA.status_Open )
      wire#w3
      { S7_Templates := "SrcType := Real" } GT_Contact(in1 := #DYNAMIC_DATA.actual_Runon_Timer, in2 := 0.0)
   END_RUNG wire#w2
   RUNG wire#w3
      Contact( #STATIC_DATA.CONFIG_MAINT_OP )
   END_RUNG wire#w2
   RUNG wire#w2
      Coil( #DYNAMIC_DATA.status_OpenOn )
   END_RUNG
   // the same network as SCL:
   #OPEN_CMD := NOT #wrkCtrlPriority40 AND NOT #DYNAMIC_DATA.status_Fault AND #DYNAMIC_DATA."$ctrl_OpenClose" AND (#DYNAMIC_DATA.status_Opening OR (#DYNAMIC_DATA.status_Open AND ((#DYNAMIC_DATA.actual_Runon_Timer > 0.0) OR #STATIC_DATA.CONFIG_MAINT_OP)));
   #DYNAMIC_DATA.status_OpenOn := #OPEN_CMD;
END_REGION

REGION Network 48: CLOSE_CMD output driver
   // ▀▀▀▀▀▀▀▀▀▀▀▀▀▀▀▀▀▀▀▀▀▀▀▀▀▀▀▀▀▀▀▀▀▀▀▀▀▀▀▀▀▀▀▀
   // The OPEN_CMD output drive will activate if all the following are true:
   // 
   //    1.  ESTOP is healthy or disabled (#wrkCtrlPriority40 = 1)
   // 
   //    2.  There is no fault condition (status_Fault = 0)
   // 
   //    3.  The valve is requested closed ($ctrl_OpenClose = 0)
   // 
   //    4. The valve is closing (status_Closing =1)
   //         OR
   //      The valve is closed (status_Closed = 1) and either the run-on timer is active
   //      or the valve is configured to maintain outputs (CONFIG_MAINT_OP = 1)
   // 
   // The status_CloseOn signal is set to match the state of the CLOSE_CMD
   // ▄▄▄▄▄▄▄▄▄▄▄▄▄▄▄▄▄▄▄▄▄▄▄▄▄▄▄▄▄▄▄▄▄▄▄▄▄▄▄▄▄▄▄▄
   RUNG wire#powerrail
      I_Contact( #wrkCtrlPriority40 )
      I_Contact( #DYNAMIC_DATA.status_Fault )
      I_Contact( #DYNAMIC_DATA."$ctrl_OpenClose" )
      wire#w1
      Contact( #DYNAMIC_DATA.status_Closing )
      wire#w2
      Coil( #CLOSE_CMD )
   END_RUNG
   RUNG wire#w1
      Contact( #DYNAMIC_DATA.status_Closed )
      wire#w3
      { S7_Templates := "SrcType := Real" } GT_Contact(in1 := #DYNAMIC_DATA.actual_Runon_Timer, in2 := 0.0)
   END_RUNG wire#w2
   RUNG wire#w3
      Contact( #STATIC_DATA.CONFIG_MAINT_OP )
   END_RUNG wire#w2
   RUNG wire#w2
      Coil( #DYNAMIC_DATA.status_CloseOn )
   END_RUNG
   // the same network as SCL:
   #CLOSE_CMD := NOT #wrkCtrlPriority40 AND NOT #DYNAMIC_DATA.status_Fault AND NOT #DYNAMIC_DATA."$ctrl_OpenClose" AND (#DYNAMIC_DATA.status_Closing OR (#DYNAMIC_DATA.status_Closed AND ((#DYNAMIC_DATA.actual_Runon_Timer > 0.0) OR #STATIC_DATA.CONFIG_MAINT_OP)));
   #DYNAMIC_DATA.status_CloseOn := #CLOSE_CMD;
END_REGION

REGION Network 49: LICENCE AND CONTACT INFORMATION
   // ▀▀▀▀▀▀▀▀▀▀▀▀▀▀▀▀▀▀▀▀▀▀▀▀▀▀▀▀▀▀▀▀▀▀▀▀▀▀▀▀▀▀▀▀
   // LICENCE AND CONTACT INFORMATION
   // 
   // This software and its associated documentation is made available under the MIT Licence:
   // 
   // ════════════════════════════════════════════
   // 
   // The MIT License (MIT)
   // 
   // Copyright © 2020 Michael Gledhill
   // 
   // Permission is hereby granted, free of charge, to any person obtaining a copy of this software 
   // and associated documentation files (the “Software”), to deal in the Software without restriction, 
   // including without limitation the rights to use, copy, modify, merge, publish, distribute, 
   // sublicense, and/or sell copies of the Software, and to permit persons to whom the Software is 
   // furnished to do so, subject to the following conditions: 
   // 
   // The above copyright notice and this permission notice shall be included in all copies or 
   // substantial portions of the Software.
   // 
   // THE SOFTWARE IS PROVIDED “AS IS”, WITHOUT WARRANTY OF ANY KIND, EXPRESS OR IMPLIED, 
   // INCLUDING BUT NOT LIMITED TO THE WARRANTIES OF MERCHANTABILITY, FITNESS FOR A 
   // PARTICULAR PURPOSE AND NON-INFRINGEMENT. IN NO EVENT SHALL THE AUTHORS OR COPYRIGHT 
   // HOLDERS BE LIABLE FOR ANY CLAIM, DAMAGES OR OTHER LIABILITY, WHETHER IN AN ACTION OF 
   // CONTRACT, TORT OR OTHERWISE, ARISING FROM, OUT OF OR IN CONNECTION WITH THE SOFTWARE 
   // OR THE USE OR OTHER DEALINGS IN THE SOFTWARE.
   // 
   // ════════════════════════════════════════════
   //                    ┌────────────┐
   // You can reach the author by email here:   │  mg@practicalseries.com  │
   //                    └────────────┘
   // Questions, corrections, constructive criticism and complaints (polite ones) are invited.
   RUNG wire#powerrail
      I_Contact( #SYS_SIGNALS._False )
      wire#w1
      S_Move(in := 'MIT LICENSE', out => #licInfo.LICENCE_TYPE)
   END_RUNG
   RUNG wire#w1
      S_Move(in := '2020 Michael Gledhill', out => #licInfo.COPYRIGHT)
   END_RUNG
   // the same network as SCL:
   IF NOT #SYS_SIGNALS._False THEN
       #licInfo.LICENCE_TYPE := 'MIT LICENSE';
       #licInfo.COPYRIGHT := '2020 Michael Gledhill';
   END_IF;
END_REGION
END_FUNCTION
